// TIA Portal V20 export
// export: Created 2025-12-01T14:57:13.6851752Z, ExportSetting None, DisplayName Totally Integrated Automation Portal, DisplayVersion V20 Update 3, DisplayName TIA Portal Openness, DisplayVersion V20 Update 3, DisplayName TIA Portal Version Control Interface, DisplayVersion V20 Update 3, DisplayName STEP 7 Professional, DisplayVersion V20 Update 3, DisplayName STEP 7 Safety, DisplayVersion V20 Update 2, DisplayName WinCC Basic/Comfort/Advanced, DisplayVersion V20 Update 3, DisplayName WinCC Professional, DisplayVersion V20 Update 3, DisplayName WinCC Unified, DisplayVersion V20 Update 3
FUNCTION "FC804_JDT01AnalisisRecibidos" : Void   // FC804, LAD
TITLE = "AnalisisRecibidos" - Analizar los mensajes recibidos por TCP/IP
{ S7_Optimized_Access := 'FALSE' }
AUTHOR : TRACKING
NAME : 20141014
VERSION : 4.0
// - Analizar si el mensaje en si es correcto
// - Distribución
//    - Mensaje ACKN (Validar ID)
//    - Mensaje PING
//    - Resto de mensajes (Validar ID)
// stored: AutoNumber false, SetENOAutomatically false
   VAR_TEMP
      Longitud : UDInt;   // Longitud del Mensaje
      IDMensaje : UDInt;   // ID del Mensaje Recibido
      IniListaEventos : DWord;   // Puntero donde empieza la lista de los eventos
      BytesListaEventos : UDInt;   // Numero de bytes que tiene la lista de los eventos
      DBUltimoRec : Word;   // DB del Ultimo Mensaje Recibido
      DBUltimoEmi : Word;   // DB del Ultimo Mensaje Enviado
      DBEventosRec : Word;   // DB de lista de Eventos Recibidos
      DBEmiAK : Word;   // DB de Emision del Evento AK - Confirmacion
      ReturnValor : Int;   // Temporal
      POrigen : Any;   // Puntero ANY del Origen
      PDestino : Any;   // Puntero ANY del Destino
      IdentEmisor : DWord;
      IdentReceptor : DWord;
      TMPEsperaKA : UDInt;
   END_VAR
BEGIN

NETWORK
TITLE = Inicializamos
// - Inicializaciones de las variables de los DB
// - Coger de la configuracion el Identificador del Emisor (12)
// - Coger de la configuracion el Identificador del Receptor (18)
// -------------------------------------------------------------------------------------------
// Si trabaja sin Agencia  2018 01 24
      SET;
      AN    "Activar_JDT01";  // Mirar si se trabaja con agencia
      JC    Final;

// --------------------------------------------------------------------------------------------
// Inicializaciones de las variables de los DB

      L     "JDT1_NDB_UltimoRec";  // Cogemos el DB de UltimoRecibido
      T     #DBUltimoRec;
      L     "JDT1_NDB_EventosRec";  // Cogemos el DB de EventosRecibidos
      T     #DBEventosRec;

      L     "JDT1_NDB_AKEmi";  // Cogemos el DB de EmisionAK
      T     #DBEmiAK;
      L     "JDT1_NDB_UltimoEmi";  // Cogemos el DB de UltimoEnviado
      T     #DBUltimoEmi;


// --------------------------------------------------------------------------------------------
// Coger de la configuracion el Idendificador del emisor

      L     "JDT1_IdentEmisor";
      T     #IdentEmisor;

// --------------------------------------------------------------------------------------------
// Coger de la configuracion el Idendificador del receptor

      L     "JDT1_IdentReceptor";
      T     #IdentReceptor;


NETWORK
TITLE = Comprobación de la consistencia del mensaje
// Mirar si es correcto
// - Si es Inicio del Mensaje
// - Si es Fin del Mensaje
// - Si es Correcto el Destinario del Mensaje
// - Si es Correcto el Origen del Mensaje
// --------------------------------------------------------------------------------------------
// Mirar si hay mensaje

      L     0;  // Preparar el puntero al Primer byte
      LAR1;
      OPN   DB [#DBUltimoRec];
      L     DBB [AR1, P#0.0];  // Si hay mensaje a tratar <> 0 el primer byte
      L     0;
      ==I;
      JC    Final;  // No hay mensaje

// --------------------------------------------------------------------------------------------
// 1º Paso - Comprobación de que existe Inicio de Mensaje

      OPN   DB [#DBUltimoRec];
      L     DBB [AR1, P#0.0];  // Inicio de Mensaje debe ser 0x02
      L     2;
      ==I;
      JCN   ErrorDeMensajeRecibido;  // Error de Mensaje, Inicio NOK

// --------------------------------------------------------------------------------------------
// 2º Paso - Comprobación de que existe Final del Mensaje

      CALL  "FC890_EtiqChar_EtiqDInt"
      ( DB_String   := "JDT1_NDB_UltimoRec",  // DB del UltimoRecibido
        Long_String := 5,
        Offset_Ini  := 20,
        Valor       := #Longitud
      );  // Calcular la longitud del mensaje

      L     #Longitud;  // Preparar el puntero
      L     1;
      -D;
      SLD   3;
      LAR1;
      OPN   DB [#DBUltimoRec];  // Fin de Mensaje debe ser 0x03
      L     DBB [AR1, P#0.0];
      L     3;
      ==I;
      JCN   ErrorDeMensajeRecibido;  // Error de Mensaje, Fin NOK

// --------------------------------------------------------------------------------------------
// 3º Paso - Comprobación del Emisor del  Mensaje

      L     0;  // Preparar Puntero
      LAR1;
      OPN   DB [#DBUltimoRec];
      L     DBD [AR1, P#6.0];  // Comprobacion del Emisor
      L     #IdentReceptor;
      <>D;
      JC    ErrorDeMensajeRecibido;  // Error de Mensaje, Emisor NOK

// --------------------------------------------------------------------------------------------
// 4º Paso - Comprobación del Receptor del  Mensaje

      OPN   DB [#DBUltimoRec];
      L     DBD [AR1, P#11.0];  // Comprobación del Receptor
      L     #IdentEmisor;
      <>D;
      JC    ErrorDeMensajeRecibido;  // Error de Mensaje, Receptor NOK


NETWORK
TITLE = Distribucion
// - Mirar si es mensaje ACKN - Confirmacion
// - Mirar si es mensaje PING - Keep Alive
// - Es Mensaje de Evento
// --------------------------------------------------------------------------------------------
// 1º Paso - Mirar si es Mensaje AK

      L     0;  // Preparar puntero
      LAR1;
      OPN   DB [#DBUltimoRec];
      L     DBD [AR1, P#24.0];
      L     'ACKN';
      ==I;
      JC    MensajeRecibido_AcuseDeRecibo;  // Recibido Mensaje ACKN - Confirmacion

// --------------------------------------------------------------------------------------------
// 2º Paso - Mirar si es Mensaje KA

      OPN   DB [#DBUltimoRec];
      L     DBD [AR1, P#24.0];
      L     'PING';
      ==I;
      JC    MensajeRecibido_KeepAlive;  // Recibido Mensaje PING - Keep Alive

// --------------------------------------------------------------------------------------------
// 3º Paso - Es Mensaje Evento

      JU    MensajeRecibido_ListaDeEventos;  // Otro tipo de Evento


NETWORK
TITLE = Recibido Mensaje ACKN - Confirmacion del Mensaje Enviado
// - Mirar si esta esperando el Mensaje ACKN - Confirmacion
// - Comprobacion del ID del Mensaje
// - Si es el mismo Numero Secuencial dar por envioado el Mensaje
// - Resetear la variable del Timer Keep Alive y Borrar Mensaje Tratado
// --------------------------------------------------------------------------------------------
// 1º Paso - Comprobamos si esta esperando el Mensaje

MensajeRecibido_AcuseDeRecibo:NOP   0;

      L     0;
      LAR1;
      OPN   DB [#DBUltimoEmi];
      L     DBB [AR1, P#0.0];
      L     'N';  // Mirar si esta esperando que se reciba el AK
      <>I;
      JC    MensajeRecibido_Inesperado;  // No espara el Mensaje AK

// --------------------------------------------------------------------------------------------
// 2º Paso - Comprobamos ID del mensaje

      CALL  "FC890_EtiqChar_EtiqDInt"
      ( DB_String   := "JDT1_NDB_UltimoRec",  // DB del UltimoRecibido
        Long_String := 4,
        Offset_Ini  := 4,
        Valor       := #IDMensaje
      );  // Calcular  el Numero Secuencial

      L     #IDMensaje;  // Si es el mismo Numero Secuencial
      L     "DB801_JDT01StatusCOM".ID_UltimoEnviado;
      <>I;
      JC    MensajeRecibido_Inesperado;  // No es el mismo Numero Secuencial

// --------------------------------------------------------------------------------------------
// 3º Paso - Si es el mismo Numero Secuencial dar por enviado el Mensaje

      SET;
      R     "DB801_JDT01StatusCOM".EsperandoAK;
// nieves Control  reintentos
      L     0;
      T     "Reintentos_JDT1";


// fin control reintentos



      CALL  "FC898_BorrarMensaje"
      ( DB_A_RESET := "DB805_JDT01UltimoEnviado"  // ¿Hay que borrar asi?
      );  // Damos por acabado el envio del mensaje

// --------------------------------------------------------------------------------------------
// 4º Paso - Resetear variable para el Timer de Keep Alive
//         - Borrar Mensaje tratado

MensajeRecibido_Inesperado:NOP   0;

      SET;
      R     "DB801_JDT01StatusCOM".KeepAlive_Recibido;  // Reseteamos el Timer de KeepAlive

      CALL  "FC898_BorrarMensaje"
      ( DB_A_RESET := "DB804_JDT01UltimoRecibido"  // ¿HAy que borrar asi?
      );  // Damos por acabado el mensaje recibido

      JU    Final;


NETWORK
TITLE = Recibido Mensaje PING - Keep Alive
// - Resetear variable que trata el Timer de Keep Alive
// - Borrar Mensaje Tratado

// --------------------------------------------------------------------------------------------
// 1º Paso - Resetear variable para el Timer de Keep Alive
//         - Borrar Mensaje tratado

MensajeRecibido_KeepAlive:NOP   0;

      SET;
      R     "DB801_JDT01StatusCOM".KeepAlive_Recibido;  // Reseteamos el Timer de KeepAlive

      CALL  "FC898_BorrarMensaje"
      ( DB_A_RESET := "DB804_JDT01UltimoRecibido"  // ¿HAy que borrar asi?
      );  // Damos por acabado el envio del mensaje

      JU    Final;



NETWORK
TITLE = Recibido Mensaje de Lista de Eventos
// - Validar el ID del Mensaje Recibido
// - Miramos si se puede tratar el Mensaje de Eventos
// - Copiar la lista de eventos
// --------------------------------------------------------------------------------------------
// 1º Paso - Validar el ID del Mensaje Recibido

MensajeRecibido_ListaDeEventos:NOP   0;

      CALL  "FC890_EtiqChar_EtiqDInt"
      ( DB_String   := "JDT1_NDB_UltimoRec",  // DB del UltimoRecibido
        Long_String := 4,
        Offset_Ini  := 4,
        Valor       := #IDMensaje
      );  // Calcular  el Numero Secuencial

      L     #IDMensaje;  // Comprobar Si el ID = 0
      L     0;
      ==I;
      JC    EINI;

      L     #IDMensaje;  // Comprobar si es el ID Valido
      L     "DB801_JDT01StatusCOM".ID_UltimoRecibido;
      ==I;
      JC    MensajeRecibido_OK;  // No es valido el Numero Secuencial, Enviar ACKN

// --------------------------------------------------------------------------------------------
// 2º Paso - Miramos si se puede tratar el Mensaje de Eventos

EINI: L     0;
      LAR1;
      OPN   DB [#DBEventosRec];
      L     DBB [AR1, P#0.0];  // Vacio - Primer Byte a 0
      L     0;
      <>I;
      JC    Final;  // No puede ser tratado todabia

// --------------------------------------------------------------------------------------------
// 3º Paso - Copiar la lista de eventos

      L     0;  // Preparo el Inicio de la Lista Eventos a Copiar
      LAR1;
      +AR1  P#22.0;
      TAR1;
      T     #IniListaEventos;

      L     #Longitud;  // Numero de Bytes de la Lista de Eventos a Copiar
      L     22;
      -D;
      T     #BytesListaEventos;

      CALL  "FC897_Generar_PointerAny"
      ( TYP           := 16#10,
        DataTyp       := 16#02,
        repeatcounter := #BytesListaEventos,  // Tamaño del mensaje
        DB_Number     := "JDT1_NDB_UltimoRec",  // DB UltimoRecibido
        storearea     := 16#84,
        storeaddresse := #IniListaEventos,
        Any_Pointer   := #POrigen
      );  // Puntero Origen

      CALL  "FC897_Generar_PointerAny"
      ( TYP           := 16#10,
        DataTyp       := 16#02,
        repeatcounter := #BytesListaEventos,  // Tamaño del mensaje
        DB_Number     := "JDT1_NDB_EventosRec",  // DB EventosRecibidos
        storearea     := 16#84,
        storeaddresse := 16#0000_0000,
        Any_Pointer   := #PDestino
      );  //Puntero Destino

      CALL  BLKMOV
      ( SRCBLK  := #POrigen,
        RET_VAL := #ReturnValor,
        DSTBLK  := #PDestino
      );  // Realizo la transferencia

      JU    MensajeRecibido_OK;



NETWORK
TITLE = Envio del Mensaje ACKN - Acuse de Recibo
// Confirmacion del Mensaje Recibido: Lista de Eventos
// -
// --------------------------------------------------------------------------------------------
// 1º Paso - Guardamos el ID del Mensaje Tratado

MensajeRecibido_OK:NOP   0;

      L     #IDMensaje;  // Guardo el ID del Mensaje Tratado
      T     "DB801_JDT01StatusCOM".ID_UltimoRecibido;

// --------------------------------------------------------------------------------------------
// 2º Paso - Formatear el Mensaje AK en e DB MensajeAK
//    - Rellenar Cabecera
//    - Rellenar Cuerpo

// Rellenar el Campo del ID del Mensaje

      CALL  "FC891_EtiqDInt_EtiqChar"
      ( DB_String   := "JDT1_NDB_AKEmi",  // DB EmisionAK
        Long_String := 4,
        Offset_Ini  := 4,
        Valor       := #IDMensaje
      );

// Preparamos Puntero DB EmisionAK
      L     0;
      LAR1;

// Rellenamos la cabecera del mensaje
      OPN   DB [#DBEmiAK];
      L     2;  // Primer Byte 0x02 - Para que sea enviada
      T     DBB [AR1, P#0.0];
      L     ';';  // Separador
      T     DBB [AR1, P#5.0];

      L     #IdentEmisor;  // Rellenar el Campo Emisor
      T     DBD [AR1, P#6.0];

      L     ';';  // Separador
      T     DBB [AR1, P#10.0];

      L     #IdentReceptor;  // Rellenar el Campo Receptor
      T     DBD [AR1, P#11.0];

      L     ';';  // Separador
      T     DBB [AR1, P#15.0];
      L     '0';  // Tamaño del Mensaje 38
      T     DBB [AR1, P#16.0];
      L     '0038';
      T     DBD [AR1, P#17.0];
      L     ';';  // Separador
      T     DBB [AR1, P#21.0];

// Rellenamos el Evento a escribir- ({ACKN[RSLT]0})
      L     '({';  // Empieza Evento
      T     DBW [AR1, P#22.0];
      L     'ACKN';  // Evento ACKN
      T     DBD [AR1, P#24.0];

      L     '[';  // Atributo del Evento RSLT
      T     DBB [AR1, P#28.0];
      L     'RSLT';  // Atributo del Evento RSLT
      T     DBD [AR1, P#29.0];
      L     ']';  // Atributo del Evento RSLT
      T     DBB [AR1, P#33.0];

      L     '0';  // Contestacion del Atributo del Evento AK
      T     DBB [AR1, P#34.0];
      L     '})';  // Final del Evento
      T     DBW [AR1, P#35.0];

// Rellenamos el final del Evento
      L     3;  // Final del Mensaje 0x03
      T     DBB [AR1, P#37.0];

// --------------------------------------------------------------------------------------------
// 3º Paso - Resetear variable para el Timer de Keep Alive
//         - Borrar Mensaje tratado

      SET;
      R     "DB801_JDT01StatusCOM".KeepAlive_Recibido;  // Reseteamos el Timer de KeepAlive

      CALL  "FC898_BorrarMensaje"
      ( DB_A_RESET := "DB804_JDT01UltimoRecibido"  // ¿HAy que borrar asi?
      );  // Damos por acabado el mensaje recibido

      JU    Final;


NETWORK
TITLE = Error del Mensaje, Mal formateado
// - Se da por tratado el mensaje, borrar
//-----------------------------------------------------------------------------------------------
// Error de mensaje, mal formateado

ErrorDeMensajeRecibido:NOP   0;
      CALL  "FC898_BorrarMensaje"
      ( DB_A_RESET := "DB804_JDT01UltimoRecibido"  // ¿Hay que Borrar todo?
      );  // Damos por acabado el Mensaje Recibido

      JU    Final;

NETWORK
TITLE = Finalizar
// Se Acabo la funcion
// - Control del temporizador KA (Reseteo)
// - Volver a Activar el temporizador KA

Final:NOP   0;

//-----------------------------------------------------------------------------------------------
// Paso 1º- Control del temporizador KA

      L     "JDT1_TMPEsperaKA";
      T     #TMPEsperaKA;
      CALL  "FC899_TMP"
      ( Temporizar     := "DB801_JDT01StatusCOM".KeepAlive_Recibido,
        Valor_Tiempo   := #TMPEsperaKA,  // TMP Espera de Recepción de KA
        Base_tiempo_ms := 1000,
        Tiempo_OK      := "DB801_JDT01StatusCOM".TMPEsperaKA_OK,
        Valor_Actual   := "DB801_JDT01StatusCOM".TMPEsperaKA  // Tiempo de 2M
      );

//-----------------------------------------------------------------------------------------------
// Paso 2º - Volver el Temporizador KA, Variable KeepAlive_Recibido = 1

      AN    "DB801_JDT01StatusCOM".KeepAlive_Recibido;
      S     "DB801_JDT01StatusCOM".KeepAlive_Recibido;

END_FUNCTION
